// TwinCAT 3 PLC project LabExercise
// ProgramVersion: 3.1.4023.0
// libraries:
//   Tc2_NCI, * (Beckhoff Automation GmbH)
//   Tc2_Standard, * (Beckhoff Automation GmbH)
//   Tc2_System, * (Beckhoff Automation GmbH)
//   Tc3_Module, * (Beckhoff Automation GmbH)
//   VisuDialogs, * (System)
// project tree:
//   Comissioning/Function blocks/ FB_ModifyAutomaticControlSettings.TcPOU (not stored)
//   Comissioning/GVLs/ G_Commissioning.TcGVL (not stored)
//   Comissioning/Struct/ ST_AutomaticControlSettings.TcDUT (not stored), ST_ClosedLoopControlSettings.TcDUT (not stored), ST_MotionReferenceGeneratorSettings.TcDUT (not stored), ST_OpenLoopControlSettings.TcDUT (not stored)
//   ControlBox/Interfaces/ I_ControlBox.TcIO (not stored)
//   ControlBox/Function blocks/ FB_ControlBox.TcPOU (not stored), FB_RealControlBox.TcPOU (not stored), FB_VirtualControlBox.TcPOU (not stored)
//   CraneControl/Function blocks/Sub blocks/ FB_ActiveDamping.TcPOU (not stored), FB_Clock.TcPOU (not stored), FB_ClosedLoopControl.TcPOU (not stored), FB_Joystick.TcPOU (not stored), FB_MotionReferenceGenerator_limit.TcPOU (not stored), FB_OpenLoopControl.TcPOU (not stored), FB_ResetIntegralController.TcPOU (not stored), FB_Status.TcPOU (not stored)
//   CraneControl/Enums/ E_Mode.TcDUT (not stored), E_Status.TcDUT (not stored)
//   CraneControl/Function blocks/Main blocks/ FB_AutomaticControl.TcPOU (not stored), FB_ManualControl.TcPOU (not stored)
//   CraneControl/Functions/ F_BarToEng.TcPOU (not stored), F_LminToEng.TcPOU (not stored), F_RadToDeg.TcPOU (not stored)
//   CraneControl/GVLs/ G_Parameters.TcGVL (not stored), G_Work.TcGVL (not stored)
//   CraneControl/Struct/ ST_ActiveDamping.TcDUT (not stored), ST_Parameters.TcDUT (not stored)
//   / GlobalTextList.TcGTLO (not stored), PlcTask.TcTTO (not stored), Simulator.TcTTO (not stored), Visualization Manager.TcVMO (not stored)
//   HMI/ HMI.TcVIS (not stored)
//   HMI/Sub/ CommissioningHMI.TcVIS (not stored), VirtualControlBox.TcVIS (not stored)
//   Inputs/ FB_JoystickInputScaling.TcPOU (not stored), FB_PositionInputScaling.TcPOU (not stored), FB_PressureInputScaling.TcPOU (not stored), G_Inputs.TcGVL (not stored), G_Sensors.TcGVL (not stored), FB_Vctrl.TcPOU
//   Inputs/Struct/ ST_AnalogInput.TcDUT (not stored), ST_AnalogInputStatus.TcDUT (not stored)
//   Outputs/ FB_ValveOutput.TcPOU (not stored), G_Outputs.TcGVL (not stored)
//   Outputs/Struct/ ST_pValveDeadBand.TcDUT (not stored), ST_ValveOutput.TcDUT (not stored)
//   ControlBox/GVLs/ G_VirtualControlBox.TcGVL (not stored)
//   Programs/ MAIN.TcPOU (not stored), P_Commissioning.TcPOU (not stored), P_ControlBox.TcPOU (not stored), P_CraneControl.TcPOU (not stored), P_Inputs.TcPOU (not stored), P_Outputs.TcPOU (not stored), P_Simulator.TcPOU (not stored)
//   Simulator/ FB_CraneSimulator.TcPOU (not stored), G_Simulator.TcGVL (not stored)
// real-time tasks:
//   TASK PlcTask: cycle T#1ms, priority 20, ADS port 350
//   TASK Simulator: cycle T#100us, priority 1, ADS port 351
// I/O:
//   DEVICE PLC (EtherCAT) (disabled), AmsNetId 5.80.90.242.2.1
//     PLC Rack (EK1200) [EK1200-5000 EtherCAT Power supply (2A E-Bus)]
//       DI (EL1008) [EL1008 8Ch. Dig. Input 24V, 3ms]
//       DO (EL2008) [EL2008 8Ch. Dig. Output 24V, 0.5A]
//       End Cap 4 (EL9011) [EL9011 End Terminal]
//   DEVICE RIO (EtherCAT) (disabled), AmsNetId 5.80.90.242.5.1
//     RIO (EK1100) [EK1100 EtherCAT Coupler (2A E-Bus)]
//       DI (EL1008) [EL1008 8Ch. Dig. Input 24V, 3ms]
//       DO (EL2008) [EL2008 8Ch. Dig. Output 24V, 0.5A]
//       AI1 (EL3068) [EL3068 8Ch. Ana. Input 0-10V]
//       AI2 (EL3068) [EL3068 8Ch. Ana. Input 0-10V]
//       AI3 (EL3174) [EL3174 4Ch. Ana. Input +/-10V Diff., +/-20mA SingleEnded, 16 Bit]
//       AO (EL4104) [EL4104 4Ch. Ana. Output 0-10V, 16bit]
//       End Cap (EL9011) [EL9011 End Terminal]
// variable links:
//   LabExercise/LabExercise Instance <-> PLC (EtherCAT)/PLC Rack (EK1200)/DI (EL1008)
//     PlcTask Inputs/G_Inputs.bTest <-> Channel 1/Input
//   LabExercise/LabExercise Instance <-> PLC (EtherCAT)/PLC Rack (EK1200)/DO (EL2008)
//     PlcTask Outputs/G_Outputs.bTest <-> Channel 1/Output
//   LabExercise/LabExercise Instance <-> RIO (EtherCAT)/RIO (EK1100)/AI1 (EL3068)
//     PlcTask Inputs/G_Inputs.stCylPos.nValue <-> AI Standard Channel 3/Value
//     PlcTask Inputs/G_Inputs.stCylPos.stStatus <-> AI Standard Channel 3/Status
//     PlcTask Inputs/G_Inputs.stJoyX.nValue <-> AI Standard Channel 1/Value
//     PlcTask Inputs/G_Inputs.stJoyX.stStatus <-> AI Standard Channel 1/Status
//     PlcTask Inputs/G_Inputs.stJoyY.nValue <-> AI Standard Channel 2/Value
//     PlcTask Inputs/G_Inputs.stJoyY.stStatus <-> AI Standard Channel 2/Status
//     PlcTask Inputs/G_Inputs.stSpoolPos.nValue <-> AI Standard Channel 4/Value
//     PlcTask Inputs/G_Inputs.stSpoolPos.stStatus <-> AI Standard Channel 4/Status
//   LabExercise/LabExercise Instance <-> RIO (EtherCAT)/RIO (EK1100)/AI2 (EL3068)
//     PlcTask Inputs/G_Inputs.stPressureCompensator.nValue <-> AI Standard Channel 3/Value
//     PlcTask Inputs/G_Inputs.stPressureCompensator.stStatus <-> AI Standard Channel 3/Status
//     PlcTask Inputs/G_Inputs.stPressureLhvSide.nValue <-> AI Standard Channel 5/Value
//     PlcTask Inputs/G_Inputs.stPressureLhvSide.stStatus <-> AI Standard Channel 5/Status
//     PlcTask Inputs/G_Inputs.stPressurePistonSide.nValue <-> AI Standard Channel 4/Value
//     PlcTask Inputs/G_Inputs.stPressurePistonSide.stStatus <-> AI Standard Channel 4/Status
//     PlcTask Inputs/G_Inputs.stPressureReturn.nValue <-> AI Standard Channel 2/Value
//     PlcTask Inputs/G_Inputs.stPressureReturn.stStatus <-> AI Standard Channel 2/Status
//     PlcTask Inputs/G_Inputs.stPressureRodSide.nValue <-> AI Standard Channel 6/Value
//     PlcTask Inputs/G_Inputs.stPressureRodSide.stStatus <-> AI Standard Channel 6/Status
//     PlcTask Inputs/G_Inputs.stPressureSupply.nValue <-> AI Standard Channel 1/Value
//     PlcTask Inputs/G_Inputs.stPressureSupply.stStatus <-> AI Standard Channel 1/Status
//   LabExercise/LabExercise Instance <-> RIO (EtherCAT)/RIO (EK1100)/AI3 (EL3174)
//     PlcTask Inputs/G_Inputs.stFlowReturnSide.nValue <-> AI Standard Channel 1/Value
//     PlcTask Inputs/G_Inputs.stFlowReturnSide.stStatus <-> AI Standard Channel 1/Status
//   LabExercise/LabExercise Instance <-> RIO (EtherCAT)/RIO (EK1100)/AO (EL4104)
//     PlcTask Outputs/G_Outputs.stValveOutput.nValveOutput <-> AO Output Channel 1/Analog output
//   LabExercise/LabExercise Instance <-> RIO (EtherCAT)/RIO (EK1100)/DI (EL1008)
//     PlcTask Inputs/G_Inputs.bAutoModeSelector <-> Channel 1/Input
//     PlcTask Inputs/G_Inputs.bManualModeSelector <-> Channel 2/Input
//     PlcTask Inputs/G_Inputs.bStartButton <-> Channel 3/Input
//     PlcTask Inputs/G_Inputs.bStopButton <-> Channel 4/Input
//   LabExercise/LabExercise Instance <-> RIO (EtherCAT)/RIO (EK1100)/DO (EL2008)
//     PlcTask Outputs/G_Outputs.bGreenLight <-> Channel 1/Output
//     PlcTask Outputs/G_Outputs.bRedLight <-> Channel 2/Output
//     PlcTask Outputs/G_Outputs.stValveOutput.bEnable <-> Channel 3/Output

// ---- Inputs/FB_Vctrl.TcPOU
FUNCTION_BLOCK FB_Vctrl
VAR_INPUT
	fbPressureInputScaling : FB_PressureInputScaling;
	nPressurePistonSide: LREAL;
    nPressureRodSide: LREAL;
    nPressureSupply: LREAL;
    nWantedSpeed: LREAL;
END_VAR
VAR_OUTPUT
    u: LREAL;
    k: LREAL;
END_VAR
VAR_TEMP
    Q: LREAL;
	nDirSwitch: LREAL;
END_VAR
END_FUNCTION_BLOCK


IF nWantedSpeed > 0.0 THEN 
	nDirSwitch := nPressurePistonSide;

	Q := nWantedSpeed * 0.00331;

ELSE 
	nDirSwitch := nPressureRodSide;
	IF nWantedSpeed < 0.0 THEN 
		Q := nWantedSpeed * 0.00236003;
	ELSE 
		Q := 0.0;
	END_IF;
END_IF;

u := ((((SQRT(700000.0 / (nPressureSupply - nDirSwitch)) * Q) * 60000.0) * 0.248) + 0.8) / 7.0;

k := Q * 60000.0;

END_FUNCTION_BLOCK
